{attribute 'GeneratedUsingTerminal: EL2595-0000-0018'}
{attribute addProperty BoxType "EL2595-0000-0018"}
{attribute addProperty Id "DOX_StatusAT %I*DOX_Status_AED8A12A6DOX_ControlAT %Q*DOX_Control_75D5C9E23WcStateAT %I*WcState_9091E0EB2InfoDataAT %I*InfoData_94A18F5E2"}
{attribute addProperty CRC "3380204062"}
{attribute addProperty Size "13"}
TYPE EL2595_C979D21E EXTENDS EtcSlaveTerminalBase_947E5A46 :
STRUCT
	{attribute addProperty Name "DOX_Status"}
	DOX_Status : DOX_Status_AED8A12A;
	{attribute addProperty Name "DOX_Control"}
	DOX_Control : DOX_Control_75D5C9E2;
	{attribute addProperty Name "WcState"}
	WcState : WcState_9091E0EB;
	{attribute addProperty Name "InfoData"}
	InfoData : InfoData_94A18F5E;
END_STRUCT
END_TYPE

(* stored: Version 1.2.0.0, ProductVersion 3.1.4024.9
   DUT EL2595_C979D21E: Id {c2798eac-f6b5-4725-ac42-c509be9c6eff} *)
